# EPICS autosave request: softGlueApp/Db/DEMUX2_settings.req
$(P)$(H)DEMUX2-$(N)_IN_Signal
$(P)$(H)DEMUX2-$(N)_OUT0_Signal
$(P)$(H)DEMUX2-$(N)_OUT1_Signal
$(P)$(H)DEMUX2-$(N)_SEL_Signal
